SUBAPPLICATION AuxInput_Schneidwerk_UP (* Subapplication Type *)
  (* Standard: 61499-2 *)
  (* Version 1.0, 2023-02-06, franz *)
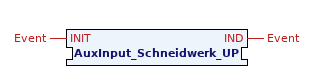
  EVENT_INPUT
    INIT;
  END_EVENT
  EVENT_OUTPUT
    IND;
  END_EVENT
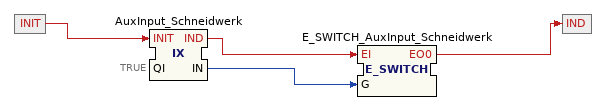
  FBS
    E_SWITCH_AuxInput_Schneidwerk : E_SWITCH;
    AuxInput_Schneidwerk : IX(QI := TRUE);
  END_FBS
  EVENT_CONNECTIONS
    AuxInput_Schneidwerk.IND TO E_SWITCH_AuxInput_Schneidwerk.EI;
    INIT TO AuxInput_Schneidwerk.INIT;
    E_SWITCH_AuxInput_Schneidwerk.EO0 TO IND;
  END_CONNECTIONS
  DATA_CONNECTIONS
    AuxInput_Schneidwerk.IN TO E_SWITCH_AuxInput_Schneidwerk.G;
  END_CONNECTIONS
END_SUBAPPLICATION
